// TIA Portal V19 export
FUNCTION "A0302_Manipolatore_CALL" : Void   // FC139, LAD
// stored: SetENOAutomatically false
   VAR_TEMP
      Missing_Input : Bool;
      Missing_Output : Bool;
   END_VAR
BEGIN

REGION Network 1: <<< CIn >>>
END_REGION

REGION Network 2 (SCL): CIn - Trasferimento stati
   // TRASFERIMENTO COMANDI CIn MANAGER
   // 
   "A0302_Manipolatore".CIn.Manager.EnableStopDoorOpeningReq := "A0302_Manager".COut.Manipolatori.Ax.EnableStopDoorOpeningReq;
   "A0302_Manipolatore".CIn.Manager.EnableStopInPhase := "A0302_Manager".COut.Manipolatori.Ax.EnableStopInPhase;
   "A0302_Manipolatore".CIn.Manager.EnableStopProgrammed := "A0302_Manager".COut.Manipolatori.Ax.EnableStopProgrammed;
   "A0302_Manipolatore".CIn.Manager.Control_ON := "A0302_Manager".COut.Manipolatori.Ax.Control_ON;
   "A0302_Manipolatore".CIn.Manager.MoveToPos := "A0302_Manager".COut.Manipolatori.Ax.MoveToPos;
   "A0302_Manipolatore".CIn.Manager.Pos := "A0302_Manager".COut.Manipolatori.Ax.Pos;
   "A0302_Manipolatore".CIn.Manager.Vel := "A0302_Manager".COut.Manipolatori.Ax.Vel;
   "A0302_Manipolatore".CIn.Manager.Acc := "A0302_Manager".COut.Manipolatori.Ax.Acc;
   "A0302_Manipolatore".CIn.Manager.Dec := "A0302_Manager".COut.Manipolatori.Ax.Dec;

   "A0302_Manipolatore".CIn.Manager.Sollevamento := "A0302_Manager".COut.Manipolatori.Sollevatori;
   "A0302_Manipolatore".CIn.Manager.Magneti := "A0302_Manager".COut.Manipolatori.Magneti;



   "A0302_Manipolatore".CIn.OP_SemiAut_PB := "A0302_Manager".DataIn.SemiAut_Pb;


   REGION TRASFERIMENTO STATI CIn ALTRE STAZIONI

       // RULLIERA
       "A0302_Manipolatore".CIn.Rulliera.Centratori := "A0302_Centratori".COut.Centratori;
       "A0302_Manipolatore".CIn.Rulliera.Coda.Sens.FTC_Rall := "A0302_Rulliera".IEC_FTC_CodaRall.FTC_On;
       "A0302_Manipolatore".CIn.Rulliera.Coda.Sens.FTC_Prox_Ing := "A0302_Rulliera".IEC_FTC_CodaProxIng.FTC_On;
       "A0302_Manipolatore".CIn.Rulliera.Centro.Sens.FTC_Centrale := "A0302_Rulliera".IEC_FTC_Centro.FTC_On;

       // CARRO PAREGGIATORE TESTA
       "A0302_Manipolatore".CIn.CarroPareggTesta.Sens.FTC1_Rall := "A0302_PareggiatoreTesta".IEC_FTC_Rall.FTC_On;
       "A0302_Manipolatore".CIn.CarroPareggTesta.Sens.FTC2_Prox_Ls := "A0302_PareggiatoreTesta".IEC_FTC_ProxLs.FTC_On;
       "A0302_Manipolatore".CIn.CarroPareggTesta.Sens.PresenzaMat := "A0302_PareggiatoreTesta".IEC_FTC_PresentMat.FTC_On;

       // CARRO PAREGGIATORE DI CODA
       "A0302_Manipolatore".CIn.CarroPareggCoda.Sens.FTC_Ingombro_In := "A0302_PareggiatoreCoda".IEC_FTC_Input.FTC_On;
       "A0302_Manipolatore".CIn.CarroPareggCoda.Sens.FTC_Ingombro_Out := "A0302_PareggiatoreCoda".IEC_FTC_Output.FTC_On;
       "A0302_Manipolatore".CIn.CarroPareggCoda.Sens.PresenzaMat := "A0302_PareggiatoreCoda".IEC_FTC_PresentMat.FTC_On;

       // STATI DELLA STAZIONE 
       "A0302_Manipolatore".CIn.CarriPareggiatori.ZoneA0302Entry_Empty := "A0302_Manager".Sts.BTrk.ZoneA0302Entry_Empty;
       "A0302_Manipolatore".CIn.CarriPareggiatori.ZoneA0302Exit_Empty := "A0302_Manager".Sts.BTrk.ZoneA0302Exit_Empty;
       "A0302_Manipolatore".CIn.CarriPareggiatori.RequestNewPosition := "A0302_Manager".Sts.Attrezzamento.RequestNewPosition;

       // SPALLE
       "A0302_Manipolatore".CIn.Spalle.Coda.ActualPos := "Areas_ITF".A04.A0303_SpallaCoda_Cout_Ax.ActualPosition;
       "A0302_Manipolatore".CIn.Spalle.Testa.ActualPos := "Areas_ITF".A04.A0303_SpallaTesta_Cout_Ax.ActualPosition;

   END_REGION ;
END_REGION

REGION Network 3: <<< DataIn >>>
END_REGION

REGION Network 4 (SCL): DataIn - OP e sensori
   // Sensori Banco di Controllo

   "A0302_Manipolatore".DataIn.Sens.Ls1 := "A0302_PezziAccumolo_Scivolo_2_Phc_1"; 
   "A0302_Manipolatore".DataIn.Sens.Ls2 := "A0302_PezziAccumolo_Scivolo_2_Phc_2"; 
   "A0302_Manipolatore".DataIn.Sens.Ls3 := "Sys".ByPass;  // Solo predisposizione
   "A0302_Manipolatore".DataIn.Sens.Ls4 := "Sys".ByPass;  // Solo predisposizione

   // Comandi OP

   "A0302_Manipolatore".DataIn.OP_MoveToPos := "A03_HMI".MB3.Button.A0302.Manipolatore.OP_Ax.MoveToPos;
   //"A0302_Manipolatore".DataIn.Sollevamento.OP.Rest := "A03_HMI".MB3.Button.A0302.Manipolatore.OP_Sollevamento.Rest;
   //"A0302_Manipolatore".DataIn.Sollevamento.OP.Work := "A03_HMI".MB3.Button.A0302.Manipolatore.OP_Sollevamento.Work;
   //"A0302_Manipolatore".DataIn.Magneti.OP.Rest := "A03_HMI".MB3.Button.A0302.Manipolatore.OP_Magneti.Rest;
   //"A0302_Manipolatore".DataIn.Magneti.OP.Work := "A03_HMI".MB3.Button.A0302.Manipolatore.OP_Magneti.Work;
END_REGION

REGION Network 5: <<< LATO TESTA >>>
END_REGION

REGION Network 6: Data In - Ax
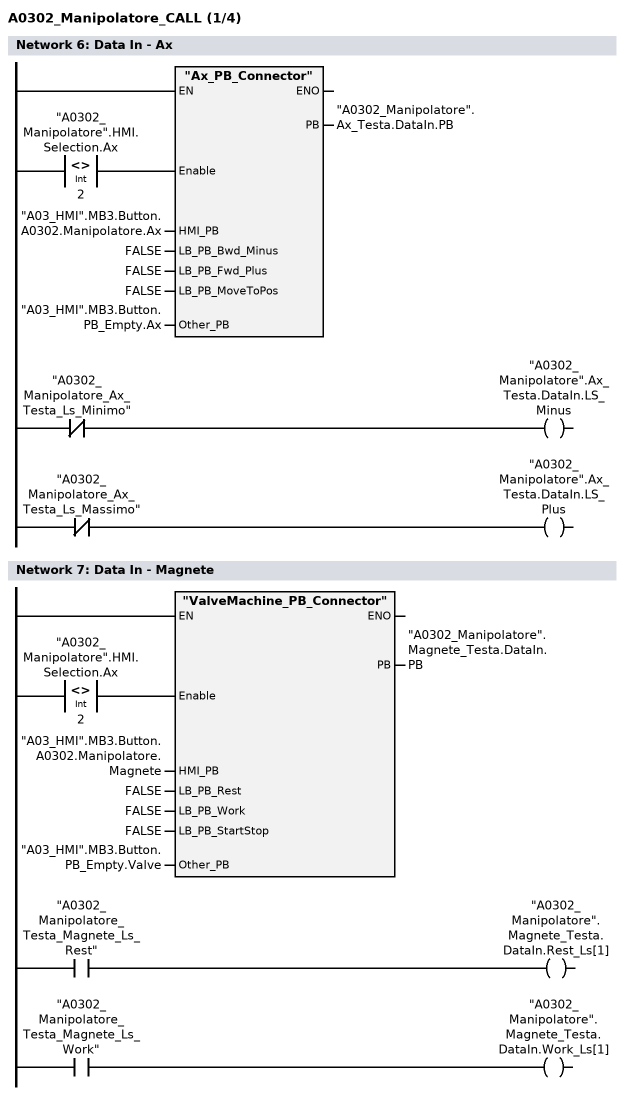
   RUNG wire#powerrail
      "Ax_PB_Connector"(Enable := wire#w1, HMI_PB := "A03_HMI".MB3.Button.A0302.Manipolatore.Ax, LB_PB_Bwd_Minus := FALSE, LB_PB_Fwd_Plus := FALSE, LB_PB_MoveToPos := FALSE, Other_PB := "A03_HMI".MB3.Button.PB_Empty.Ax, PB => "A0302_Manipolatore".Ax_Testa.DataIn.PB)
   END_RUNG
   RUNG wire#powerrail
      { S7_Templates := "SrcType := Int" } NE_Contact(in1 := "A0302_Manipolatore".HMI.Selection.Ax, in2 := 2)
   END_RUNG wire#w1
   RUNG wire#powerrail
      I_Contact( "A0302_Manipolatore_Ax_Testa_Ls_Minimo" )
      Coil( "A0302_Manipolatore".Ax_Testa.DataIn.LS_Minus )
   END_RUNG
   RUNG wire#powerrail
      I_Contact( "A0302_Manipolatore_Ax_Testa_Ls_Massimo" )
      Coil( "A0302_Manipolatore".Ax_Testa.DataIn.LS_Plus )
   END_RUNG
   // the same network as SCL:
   "Ax_PB_Connector"(Enable := "A0302_Manipolatore".HMI.Selection.Ax <> 2,
                     HMI_PB := "A03_HMI".MB3.Button.A0302.Manipolatore.Ax,
                     LB_PB_Bwd_Minus := FALSE,
                     LB_PB_Fwd_Plus := FALSE,
                     LB_PB_MoveToPos := FALSE,
                     Other_PB := "A03_HMI".MB3.Button.PB_Empty.Ax,
                     PB => "A0302_Manipolatore".Ax_Testa.DataIn.PB);
   "A0302_Manipolatore".Ax_Testa.DataIn.LS_Minus := NOT "A0302_Manipolatore_Ax_Testa_Ls_Minimo";
   "A0302_Manipolatore".Ax_Testa.DataIn.LS_Plus := NOT "A0302_Manipolatore_Ax_Testa_Ls_Massimo";
END_REGION

REGION Network 7: Data In - Magnete
   RUNG wire#powerrail
      "ValveMachine_PB_Connector"(Enable := wire#w1, HMI_PB := "A03_HMI".MB3.Button.A0302.Manipolatore.Magnete, LB_PB_Rest := FALSE, LB_PB_Work := FALSE, LB_PB_StartStop := FALSE, Other_PB := "A03_HMI".MB3.Button.PB_Empty.Valve, PB => "A0302_Manipolatore".Magnete_Testa.DataIn.PB)
   END_RUNG
   RUNG wire#powerrail
      { S7_Templates := "SrcType := Int" } NE_Contact(in1 := "A0302_Manipolatore".HMI.Selection.Ax, in2 := 2)
   END_RUNG wire#w1
   RUNG wire#powerrail
      Contact( "A0302_Manipolatore_Testa_Magnete_Ls_Rest" )
      Coil( "A0302_Manipolatore".Magnete_Testa.DataIn.Rest_Ls[1] )
   END_RUNG
   RUNG wire#powerrail
      Contact( "A0302_Manipolatore_Testa_Magnete_Ls_Work" )
      Coil( "A0302_Manipolatore".Magnete_Testa.DataIn.Work_Ls[1] )
   END_RUNG
   // the same network as SCL:
   "ValveMachine_PB_Connector"(Enable := "A0302_Manipolatore".HMI.Selection.Ax <> 2,
                           HMI_PB := "A03_HMI".MB3.Button.A0302.Manipolatore.Magnete,
                           LB_PB_Rest := FALSE,
                           LB_PB_Work := FALSE,
                           LB_PB_StartStop := FALSE,
                           Other_PB := "A03_HMI".MB3.Button.PB_Empty.Valve,
                           PB => "A0302_Manipolatore".Magnete_Testa.DataIn.PB);
   "A0302_Manipolatore".Magnete_Testa.DataIn.Rest_Ls[1] := "A0302_Manipolatore_Testa_Magnete_Ls_Rest";
   "A0302_Manipolatore".Magnete_Testa.DataIn.Work_Ls[1] := "A0302_Manipolatore_Testa_Magnete_Ls_Work";
END_REGION

REGION Network 8: Data In - Sollevatore
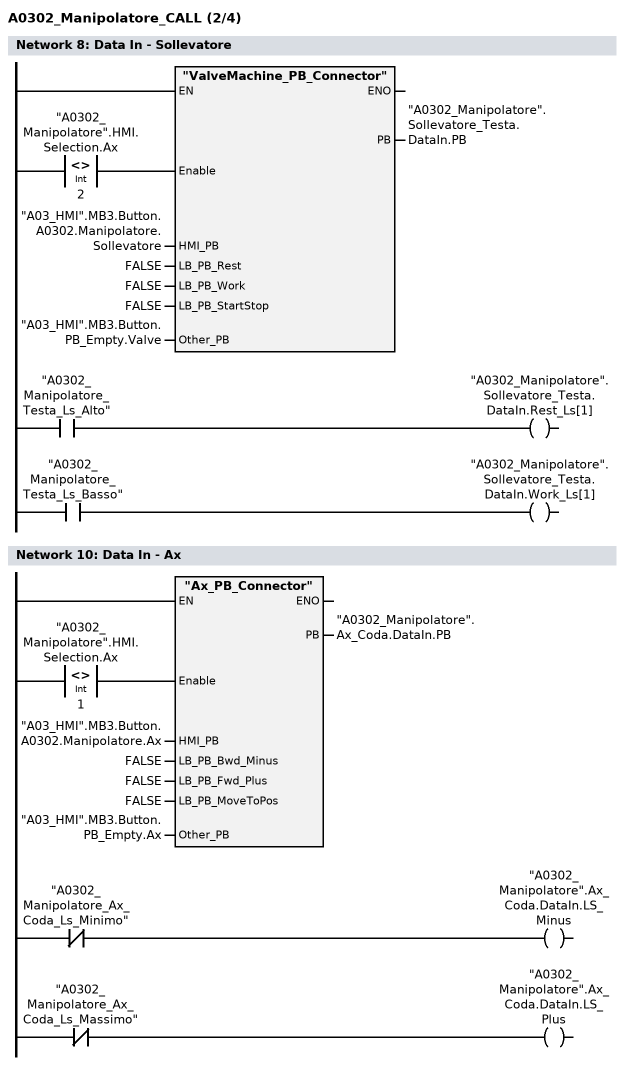
   RUNG wire#powerrail
      "ValveMachine_PB_Connector"(Enable := wire#w1, HMI_PB := "A03_HMI".MB3.Button.A0302.Manipolatore.Sollevatore, LB_PB_Rest := FALSE, LB_PB_Work := FALSE, LB_PB_StartStop := FALSE, Other_PB := "A03_HMI".MB3.Button.PB_Empty.Valve, PB => "A0302_Manipolatore".Sollevatore_Testa.DataIn.PB)
   END_RUNG
   RUNG wire#powerrail
      { S7_Templates := "SrcType := Int" } NE_Contact(in1 := "A0302_Manipolatore".HMI.Selection.Ax, in2 := 2)
   END_RUNG wire#w1
   RUNG wire#powerrail
      Contact( "A0302_Manipolatore_Testa_Ls_Alto" )
      Coil( "A0302_Manipolatore".Sollevatore_Testa.DataIn.Rest_Ls[1] )
   END_RUNG
   RUNG wire#powerrail
      Contact( "A0302_Manipolatore_Testa_Ls_Basso" )
      Coil( "A0302_Manipolatore".Sollevatore_Testa.DataIn.Work_Ls[1] )
   END_RUNG
   // the same network as SCL:
   "ValveMachine_PB_Connector"(Enable := "A0302_Manipolatore".HMI.Selection.Ax <> 2,
                           HMI_PB := "A03_HMI".MB3.Button.A0302.Manipolatore.Sollevatore,
                           LB_PB_Rest := FALSE,
                           LB_PB_Work := FALSE,
                           LB_PB_StartStop := FALSE,
                           Other_PB := "A03_HMI".MB3.Button.PB_Empty.Valve,
                           PB => "A0302_Manipolatore".Sollevatore_Testa.DataIn.PB);
   "A0302_Manipolatore".Sollevatore_Testa.DataIn.Rest_Ls[1] := "A0302_Manipolatore_Testa_Ls_Alto";
   "A0302_Manipolatore".Sollevatore_Testa.DataIn.Work_Ls[1] := "A0302_Manipolatore_Testa_Ls_Basso";
END_REGION

REGION Network 9: <<< LATO CODA >>>
END_REGION

REGION Network 10: Data In - Ax
   RUNG wire#powerrail
      "Ax_PB_Connector"(Enable := wire#w1, HMI_PB := "A03_HMI".MB3.Button.A0302.Manipolatore.Ax, LB_PB_Bwd_Minus := FALSE, LB_PB_Fwd_Plus := FALSE, LB_PB_MoveToPos := FALSE, Other_PB := "A03_HMI".MB3.Button.PB_Empty.Ax, PB => "A0302_Manipolatore".Ax_Coda.DataIn.PB)
   END_RUNG
   RUNG wire#powerrail
      { S7_Templates := "SrcType := Int" } NE_Contact(in1 := "A0302_Manipolatore".HMI.Selection.Ax, in2 := 1)
   END_RUNG wire#w1
   RUNG wire#powerrail
      I_Contact( "A0302_Manipolatore_Ax_Coda_Ls_Minimo" )
      Coil( "A0302_Manipolatore".Ax_Coda.DataIn.LS_Minus )
   END_RUNG
   RUNG wire#powerrail
      I_Contact( "A0302_Manipolatore_Ax_Coda_Ls_Massimo" )
      Coil( "A0302_Manipolatore".Ax_Coda.DataIn.LS_Plus )
   END_RUNG
   // the same network as SCL:
   "Ax_PB_Connector"(Enable := "A0302_Manipolatore".HMI.Selection.Ax <> 1,
                     HMI_PB := "A03_HMI".MB3.Button.A0302.Manipolatore.Ax,
                     LB_PB_Bwd_Minus := FALSE,
                     LB_PB_Fwd_Plus := FALSE,
                     LB_PB_MoveToPos := FALSE,
                     Other_PB := "A03_HMI".MB3.Button.PB_Empty.Ax,
                     PB => "A0302_Manipolatore".Ax_Coda.DataIn.PB);
   "A0302_Manipolatore".Ax_Coda.DataIn.LS_Minus := NOT "A0302_Manipolatore_Ax_Coda_Ls_Minimo";
   "A0302_Manipolatore".Ax_Coda.DataIn.LS_Plus := NOT "A0302_Manipolatore_Ax_Coda_Ls_Massimo";
END_REGION

REGION Network 11: Data In - Magnete
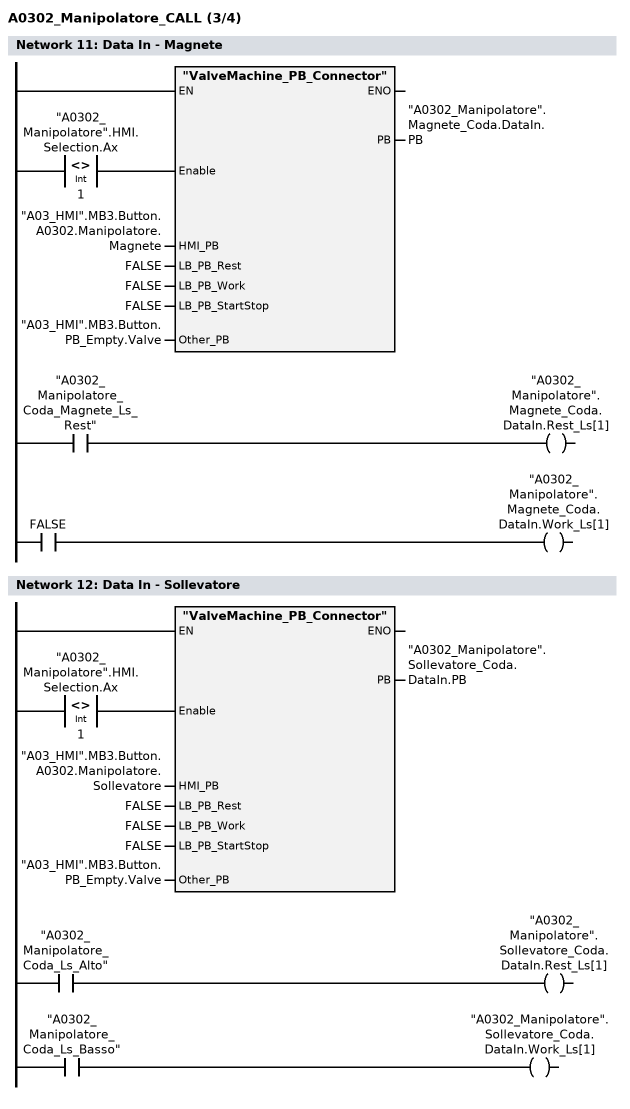
   RUNG wire#powerrail
      "ValveMachine_PB_Connector"(Enable := wire#w1, HMI_PB := "A03_HMI".MB3.Button.A0302.Manipolatore.Magnete, LB_PB_Rest := FALSE, LB_PB_Work := FALSE, LB_PB_StartStop := FALSE, Other_PB := "A03_HMI".MB3.Button.PB_Empty.Valve, PB => "A0302_Manipolatore".Magnete_Coda.DataIn.PB)
   END_RUNG
   RUNG wire#powerrail
      { S7_Templates := "SrcType := Int" } NE_Contact(in1 := "A0302_Manipolatore".HMI.Selection.Ax, in2 := 1)
   END_RUNG wire#w1
   RUNG wire#powerrail
      Contact( "A0302_Manipolatore_Coda_Magnete_Ls_Rest" )
      Coil( "A0302_Manipolatore".Magnete_Coda.DataIn.Rest_Ls[1] )
   END_RUNG
   RUNG wire#powerrail
      Contact( FALSE )
      Coil( "A0302_Manipolatore".Magnete_Coda.DataIn.Work_Ls[1] )
   END_RUNG
   // the same network as SCL:
   "ValveMachine_PB_Connector"(Enable := "A0302_Manipolatore".HMI.Selection.Ax <> 1,
                           HMI_PB := "A03_HMI".MB3.Button.A0302.Manipolatore.Magnete,
                           LB_PB_Rest := FALSE,
                           LB_PB_Work := FALSE,
                           LB_PB_StartStop := FALSE,
                           Other_PB := "A03_HMI".MB3.Button.PB_Empty.Valve,
                           PB => "A0302_Manipolatore".Magnete_Coda.DataIn.PB);
   "A0302_Manipolatore".Magnete_Coda.DataIn.Rest_Ls[1] := "A0302_Manipolatore_Coda_Magnete_Ls_Rest";
   "A0302_Manipolatore".Magnete_Coda.DataIn.Work_Ls[1] := FALSE;
END_REGION

REGION Network 12: Data In - Sollevatore
   RUNG wire#powerrail
      "ValveMachine_PB_Connector"(Enable := wire#w1, HMI_PB := "A03_HMI".MB3.Button.A0302.Manipolatore.Sollevatore, LB_PB_Rest := FALSE, LB_PB_Work := FALSE, LB_PB_StartStop := FALSE, Other_PB := "A03_HMI".MB3.Button.PB_Empty.Valve, PB => "A0302_Manipolatore".Sollevatore_Coda.DataIn.PB)
   END_RUNG
   RUNG wire#powerrail
      { S7_Templates := "SrcType := Int" } NE_Contact(in1 := "A0302_Manipolatore".HMI.Selection.Ax, in2 := 1)
   END_RUNG wire#w1
   RUNG wire#powerrail
      Contact( "A0302_Manipolatore_Coda_Ls_Alto" )
      Coil( "A0302_Manipolatore".Sollevatore_Coda.DataIn.Rest_Ls[1] )
   END_RUNG
   RUNG wire#powerrail
      Contact( "A0302_Manipolatore_Coda_Ls_Basso" )
      Coil( "A0302_Manipolatore".Sollevatore_Coda.DataIn.Work_Ls[1] )
   END_RUNG
   // the same network as SCL:
   "ValveMachine_PB_Connector"(Enable := "A0302_Manipolatore".HMI.Selection.Ax <> 1,
                           HMI_PB := "A03_HMI".MB3.Button.A0302.Manipolatore.Sollevatore,
                           LB_PB_Rest := FALSE,
                           LB_PB_Work := FALSE,
                           LB_PB_StartStop := FALSE,
                           Other_PB := "A03_HMI".MB3.Button.PB_Empty.Valve,
                           PB => "A0302_Manipolatore".Sollevatore_Coda.DataIn.PB);
   "A0302_Manipolatore".Sollevatore_Coda.DataIn.Rest_Ls[1] := "A0302_Manipolatore_Coda_Ls_Alto";
   "A0302_Manipolatore".Sollevatore_Coda.DataIn.Work_Ls[1] := "A0302_Manipolatore_Coda_Ls_Basso";
END_REGION

REGION Network 13: <+>
END_REGION

REGION Network 14 (SCL): DSI
   //
   "A0302_Manipolatore".DSI_Testa_Feed := "F_DB".DSI_ManipolatoreTesta;
   "A0302_Manipolatore".DSI_Coda_Feed := "F_DB".DSI_ManipolatoreCoda;
   "A0302_Manipolatore".DSI_Valve := "F_DB".DSI_V_Air_A0302_A0303;
END_REGION

REGION Network 15 (SCL): Drive
   "A0302_Manipolatore".Drive_Testa.Infeed_ON := "Areas_ITF".AG.Infeed_Running;
   "A0302_Manipolatore".Drive_Testa.AccessPoint := "HW_Const_Values".CU7_PN_2140A1_1_ModuleAccessPoint;
   "A0302_Manipolatore".Drive_Testa.AxisID := "CU7_ID_6_2140A1_1_2140M1";
   "A0302_Manipolatore".Drive_Testa.TokenChain := "TOKENCHAIN_CU7";

   "A0302_Manipolatore".Drive_Coda.Infeed_ON := "Areas_ITF".AG.Infeed_Running;
   "A0302_Manipolatore".Drive_Coda.AccessPoint := "HW_Const_Values".CU7_PN_2140A1_1_ModuleAccessPoint;
   "A0302_Manipolatore".Drive_Coda.AxisID := "CU7_ID_7_2140A1_2_2220M1";
   "A0302_Manipolatore".Drive_Coda.TokenChain := "TOKENCHAIN_CU7";
END_REGION

REGION Network 16 (SCL): HW
   "A0302_Manipolatore".HWID_AxTesta_TEL111 := "HW_Const_Values".CU7_PN_2140A1_1_SIEMENS_telegram_111;

   "A0302_Manipolatore".HWID_AxCoda_TEL111 := "HW_Const_Values".CU7_PN_2140A1_2_SIEMENS_telegram_111;
END_REGION

REGION Network 17: [Manipolatori] - Machine Call
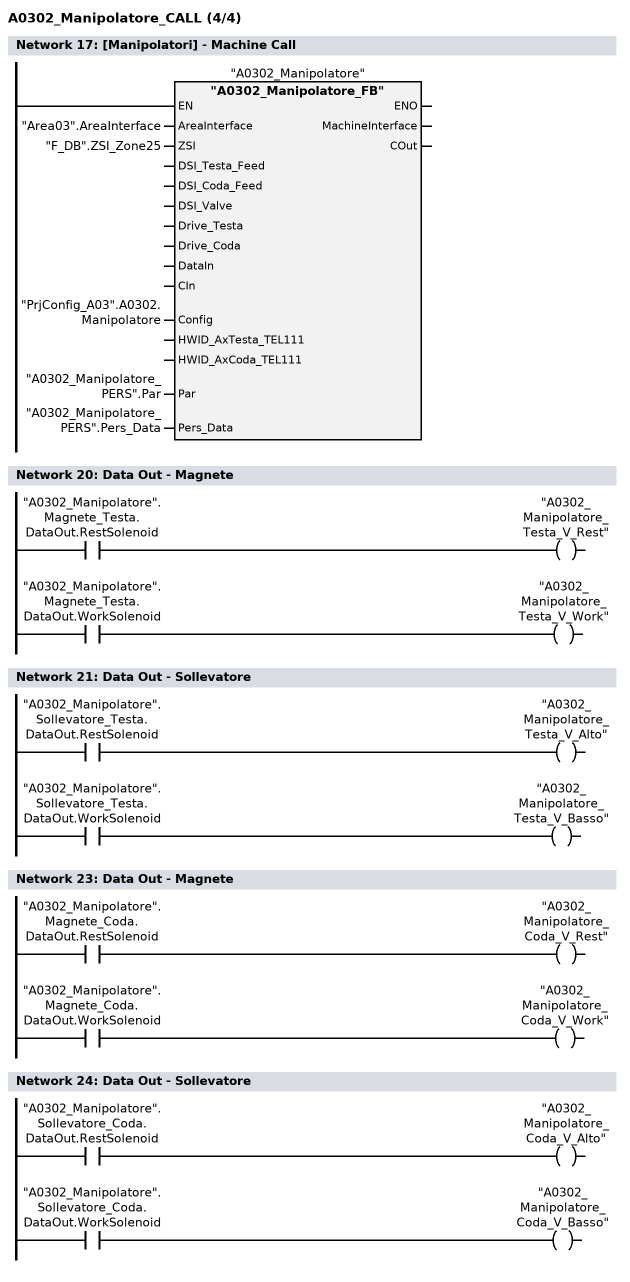
   RUNG wire#powerrail
      "A0302_Manipolatore"(AreaInterface := "Area03".AreaInterface, ZSI := "F_DB".ZSI_Zone25, DSI_Testa_Feed :=, DSI_Coda_Feed :=, DSI_Valve :=, Drive_Testa :=, Drive_Coda :=, DataIn :=, CIn :=, Config := "PrjConfig_A03".A0302.Manipolatore, HWID_AxTesta_TEL111 :=, HWID_AxCoda_TEL111 :=, Par := "A0302_Manipolatore_PERS".Par, Pers_Data := "A0302_Manipolatore_PERS".Pers_Data, MachineInterface =>, COut =>)
   END_RUNG
   // the same network as SCL:
   "A0302_Manipolatore"(AreaInterface := "Area03".AreaInterface,   // "A0302_Manipolatore_FB"
                        ZSI := "F_DB".ZSI_Zone25,
                        Config := "PrjConfig_A03".A0302.Manipolatore,
                        Par := "A0302_Manipolatore_PERS".Par,
                        Pers_Data := "A0302_Manipolatore_PERS".Pers_Data);
END_REGION

REGION Network 19: <<< LATO TESTA >>>
END_REGION

REGION Network 20: Data Out - Magnete
   RUNG wire#powerrail
      Contact( "A0302_Manipolatore".Magnete_Testa.DataOut.RestSolenoid )
      Coil( "A0302_Manipolatore_Testa_V_Rest" )
   END_RUNG
   RUNG wire#powerrail
      Contact( "A0302_Manipolatore".Magnete_Testa.DataOut.WorkSolenoid )
      Coil( "A0302_Manipolatore_Testa_V_Work" )
   END_RUNG
   // the same network as SCL:
   "A0302_Manipolatore_Testa_V_Rest" := "A0302_Manipolatore".Magnete_Testa.DataOut.RestSolenoid;
   "A0302_Manipolatore_Testa_V_Work" := "A0302_Manipolatore".Magnete_Testa.DataOut.WorkSolenoid;
END_REGION

REGION Network 21: Data Out - Sollevatore
   RUNG wire#powerrail
      Contact( "A0302_Manipolatore".Sollevatore_Testa.DataOut.RestSolenoid )
      Coil( "A0302_Manipolatore_Testa_V_Alto" )
   END_RUNG
   RUNG wire#powerrail
      Contact( "A0302_Manipolatore".Sollevatore_Testa.DataOut.WorkSolenoid )
      Coil( "A0302_Manipolatore_Testa_V_Basso" )
   END_RUNG
   // the same network as SCL:
   "A0302_Manipolatore_Testa_V_Alto" := "A0302_Manipolatore".Sollevatore_Testa.DataOut.RestSolenoid;
   "A0302_Manipolatore_Testa_V_Basso" := "A0302_Manipolatore".Sollevatore_Testa.DataOut.WorkSolenoid;
END_REGION

REGION Network 22: <<< LATO CODA >>>
END_REGION

REGION Network 23: Data Out - Magnete
   RUNG wire#powerrail
      Contact( "A0302_Manipolatore".Magnete_Coda.DataOut.RestSolenoid )
      Coil( "A0302_Manipolatore_Coda_V_Rest" )
   END_RUNG
   RUNG wire#powerrail
      Contact( "A0302_Manipolatore".Magnete_Coda.DataOut.WorkSolenoid )
      Coil( "A0302_Manipolatore_Coda_V_Work" )
   END_RUNG
   // the same network as SCL:
   "A0302_Manipolatore_Coda_V_Rest" := "A0302_Manipolatore".Magnete_Coda.DataOut.RestSolenoid;
   "A0302_Manipolatore_Coda_V_Work" := "A0302_Manipolatore".Magnete_Coda.DataOut.WorkSolenoid;
END_REGION

REGION Network 24: Data Out - Sollevatore
   RUNG wire#powerrail
      Contact( "A0302_Manipolatore".Sollevatore_Coda.DataOut.RestSolenoid )
      Coil( "A0302_Manipolatore_Coda_V_Alto" )
   END_RUNG
   RUNG wire#powerrail
      Contact( "A0302_Manipolatore".Sollevatore_Coda.DataOut.WorkSolenoid )
      Coil( "A0302_Manipolatore_Coda_V_Basso" )
   END_RUNG
   // the same network as SCL:
   "A0302_Manipolatore_Coda_V_Alto" := "A0302_Manipolatore".Sollevatore_Coda.DataOut.RestSolenoid;
   "A0302_Manipolatore_Coda_V_Basso" := "A0302_Manipolatore".Sollevatore_Coda.DataOut.WorkSolenoid;
END_REGION
END_FUNCTION
